ADAPTER ISensorStatus (* Adapter Interface *)
  (* Standard: 61499-1 *)
  (* Version 0.0, 15/09/2026 *)
  PACKAGE Hidryco.HidrycoLib;
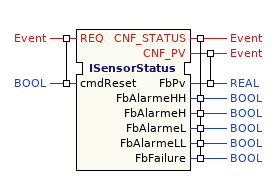
  EVENT_INPUT
    REQ WITH cmdReset; (* Request from Socket *)
  END_EVENT
  EVENT_OUTPUT
    CNF_STATUS WITH FbAlarmeHH, FbAlarmeH, FbAlarmeL, FbAlarmeLL, FbFailure; (* Confirmation from Plug *)
    CNF_PV WITH FbPv;
  END_EVENT
  VAR_INPUT
    cmdReset : BOOL;
  END_VAR
  VAR_OUTPUT
    FbPv : REAL;
    FbAlarmeHH : BOOL;
    FbAlarmeH : BOOL;
    FbAlarmeL : BOOL;
    FbAlarmeLL : BOOL;
    FbFailure : BOOL;
  END_VAR
  SERVICE SOCKET/PLUG
    SEQUENCE request_confirm
      SOCKET.REQ(REQD) -> PLUG.REQ(REQD);
      PLUG.CNF_STATUS(CNFD) -> SOCKET.CNF_STATUS(CNFD);
    END_SEQUENCE
    SEQUENCE indication_response
      PLUG.IND(INDD) -> SOCKET.IND(INDD);
      SOCKET.RSP(RSPD) -> PLUG.RSP(RSPD);
    END_SEQUENCE
  END_SERVICE
END_ADAPTER
